FUNCTION_BLOCK UsesFoo1
VAR_INPUT
    foo : REFERENCE TO Foo;
END_VAR

IF __ISVALIDREF(foo) THEN
    foo();
END_IF

END_FUNCTION_BLOCK

(* stored: Version 1.1.0.1, ProductVersion 3.1.4024.4
   POU UsesFoo1: Id {cdaa2c9d-67d7-4a5a-880f-8b044bb4e31c}, SpecialFunc None *)
